// TIA Portal V17 export
// export: Created 2025-03-05T08:00:57.341892Z, ExportSetting WithDefaults, DisplayName Totally Integrated Automation Portal, DisplayVersion V17 Update 8, DisplayName TIA Portal Openness, DisplayVersion V17 Update 8, DisplayName TIA Portal Version Control Interface, DisplayVersion V17, DisplayName SINAMICS Startdrive Advanced, DisplayVersion V17 SP2, DisplayName SINAMICS Startdrive G110M, G120, G120C, G120D, G120P, G115D, DisplayVersion V17 SP2, DisplayName SINAMICS Startdrive G130, G150, S120, S150, SINAMICS MV, S210, DisplayVersion V17 SP2, DisplayName STEP 7 Professional, DisplayVersion V17 Update 8, DisplayName SINUMERIK ONE STEP 7 Toolbox, DisplayVersion V17 Update 12, DisplayName SINUMERIK 840D sl STEP 7 Toolbox, DisplayVersion V17 Update 12, DisplayName STEP 7 Safety, DisplayVersion V17 Update 6, DisplayName WinCC Advanced, DisplayVersion V17 Update 8
FUNCTION_BLOCK "FB1501_GENERAL_GAS_SYSTEM_VALVE"   // FB1501, LAD
{ S7_Optimized_Access := 'FALSE' }
AUTHOR : ETXETAR
VERSION : 1.0
// stored: AutoNumber false, IsIECCheckEnabled false, SetENOAutomatically false, UDAEnableTagReadback false
   VAR_INPUT
      PRESSURE : Bool;   // PRESSURE INPUT
      HMI_REQ_LINE : Bool;   // HMI REQUEST LINE
   END_VAR
   VAR_OUTPUT
      HMI_POWER_UP_COND_OFF : Bool;   // HMI POWER UP CONDITIONS OFF
      HMI_POWER_UP_COND_ON : Bool;   // HMI POWER UP CONDITIONS ON
      HMI_POWER_UP_EXECU_LEFT : Bool;   // HMI POWER UP EXECUTABLE LEFT
      HMI_POWER_UP_EXECU_RIGHT : Bool;   // HMI POWER UP EXECUTABLE RIGHT
      MAIN_VALVE : Bool;   // MAIN VALVE OUTPUT
   END_VAR
   VAR DB_SPECIFIC
      AIR_FLOW_VALUE : Real;   // AIR FLOW INPUT
      TEMPERATURE_VALUE : Real;   // TEMPERATURE INPUT VALUE
      PRESS_NOT_REACHED_ALARM : Bool;   // PRESSURE NOT REACHED ALARM
      PRESS_SWITCH_ALARM : Bool;   // PRESSURE SWITCH ALARM
      PRESS_MISSING_ALARM : Bool;   // PRESSURE MISSING ALARM
      CONNECTION_SENSOR_1_ALARM : Bool;   // CONNECTION SENSOR 1 ALARM
      CONNECTION_SENSOR_2_ALARM : Bool;   // CONNECTION SENSOR 2 ALARM
      UNBLOCK_DRIVE_PRESS_ALARM : Bool;   // UNBLOCK DRIVE PRESSURE ALARM
      UNBLOCK_DRIVE_PRESS_SWITCH_ALARM : Bool;   // UNBLOCK DRIVE PRESSURE SWITCH ALARM
      PRESSURIZATION_ALARM : Bool;   // PRESSURIZATION ALARM
      PRESSURIZATION_SWITCH_ALARM : Bool;   // PRESSURIZATION SWITCH ALARM
      PNEUMATIC_TEMPERATURE_INPUT_ALARM : Bool;   // PNEUMATIC INPUT TEMPERATURE ALARM
      PNEUMATIC_FLOW_INPUT_ALARM : Bool;   // PNEUMATIC INPUT FLOW ALARM
      U01_GRIPPER_PRESSURIZATION_ALARM : Bool;   // UNIT 01 GRIPPER PRESSURIZATION ALARM
      U01_GRIPPER_PRESSURIZATION_SWITCH_ALARM : Bool;   // UNIT 01 GRIPPER PRESSURIZATION SWITCH ALARM
      U01_LABERINT_PRESSURIZATION_ALARM : Bool;   // UNIT 01 LABERINT PRESSURIZATION ALARM
      U01_LABERINT_PRESSURIZATION_SWITCH_ALARM : Bool;   // UNIT 01 LABERINT PRESSURIZATION SWITCH ALARM
      U01_UPPER_TABLE_PRESSURIZATION_ALARM : Bool;   // UNIT 01 UPPER TABLE PRESSURIZATION ALARM
      U01_UPPER_TABLE_PRESSURIZATION_SWITCH_ALARM : Bool;   // UNIT 01 UPPER TABLE PRESSURIZATION SWITCH ALARM
      U01_LOWER_TABLE_PRESSURIZATION_ALARM : Bool;   // UNIT 01 LOWER TABLE PRESSURIZATION ALARM
      U01_LOWER_TABLE_PRESSURIZATION_SWITCH_ALARM : Bool;   // UNIT 01 LOWER TABLE PRESSURIZATION SWITCH ALARM
      U01_CART_AXIS_X_PRESSURIZATION_ALARM : Bool;   // UNIT 01 CART AXIS X PRESSURIZATION ALARM
      U01_CART_AXIS_X_PRESSURIZATION_SWITCH_ALARM : Bool;   // UNIT 01 CART AXIS X PRESSURIZATION SWITCH ALARM
      U01_STA_3_MEAS_PRESSURIZATION_ALARM : Bool;   // UNIT 01 STATION 3 MEASUREMENT UNIT PRESSURIZATION ALARM
      U01_STA_3_MEAS_PRESSURIZATION_SWITCH_ALARM : Bool;   // UNIT 01 STATION 3 MEASUREMENT UNIT PRESSURIZATION SWITCH ALARM
      U02_GRIPPER_PRESSURIZATION_ALARM : Bool;   // UNIT 02 GRIPPER PRESSURIZATION ALARM
      U02_GRIPPER_PRESSURIZATION_SWITCH_ALARM : Bool;   // UNIT 02 GRIPPER PRESSURIZATION SWITCH ALARM
      U02_LABERINT_PRESSURIZATION_ALARM : Bool;   // UNIT 02 LABERINT PRESSURIZATION ALARM
      U02_LABERINT_PRESSURIZATION_SWITCH_ALARM : Bool;   // UNIT 02 LABERINT PRESSURIZATION SWITCH ALARM
      U02_UPPER_TABLE_PRESSURIZATION_ALARM : Bool;   // UNIT 02 UPPER TABLE PRESSURIZATION ALARM
      U02_UPPER_TABLE_PRESSURIZATION_SWITCH_ALARM : Bool;   // UNIT 02 UPPER TABLE PRESSURIZATION SWITCH ALARM
      U02_LOWER_TABLE_PRESSURIZATION_ALARM : Bool;   // UNIT 02 LOWER TABLE PRESSURIZATION ALARM
      U02_LOWER_TABLE_PRESSURIZATION_SWITCH_ALARM : Bool;   // UNIT 02 LOWER TABLE PRESSURIZATION SWITCH ALARM
      U02_CART_AXIS_X_PRESSURIZATION_ALARM : Bool;   // UNIT 02 CART AXIS X PRESSURIZATION ALARM
      U02_CART_AXIS_X_PRESSURIZATION_SWITCH_ALARM : Bool;   // UNIT 02 CART AXIS X PRESSURIZATION SWITCH ALARM
      U02_STA_3_MEAS_PRESSURIZATION_ALARM : Bool;   // UNIT 02 STATION 3 MEASUREMENT UNIT PRESSURIZATION ALARM
      U02_STA_3_MEAS_PRESSURIZATION_SWITCH_ALARM : Bool;   // UNIT 02 STATION 3 MEASUREMENT UNIT PRESSURIZATION SWITCH ALARM
      SWITCH_ON_GENERAL_CONDITIONS : Bool;   // SWITCH ON GENERAL CONDITIONS
      SWITCH_ON_INITIAL_CONDITIONS : Bool;   // SWITCH ON INITIAL CONDITIONS
      SWITCH_ON_MANUAL_REQUEST : Bool;   // SWITCH ON MANUAL REQUEST
      SWITCH_ON_AUTO_REQUEST : Bool;   // SWITCH ON AUTO REQUEST
      SWITCH_ON_GLOBAL_REQUEST : Bool;   // SWITCH ON GLOBAL REQUEST
      SWITCH_ON_COMMAND : Bool;   // SWITCH ON COMMAND
      SWITCH_ON : Bool;   // SWITCH ON
      IN_SERVICE : Bool;   // IN SERVICE
      SWITCH_OFF_GENERAL_CONDITIONS : Bool;   // SWITCH OFF GENERAL CONDITIONS
      SWITCH_OFF_INITIAL_CONDITIONS : Bool;   // SWITCH OFF INITIAL CONDITIONS
      SWITCH_OFF_MANUAL_REQUEST : Bool;   // SWITCH OFF MANUAL REQUEST
      SWITCH_OFF_AUTO_REQUEST : Bool;   // SWITCH OFF AUTO REQUEST
      SWITCH_OFF_GLOBAL_REQUEST : Bool;   // SWITCH OFF GLOBAL REQUEST
      SWITCH_OFF_COMMAND : Bool;   // SWITCH OFF COMMAND
      SWITCH_OFF : Bool;   // SWITCH OFF
      OUT_OF_SERVICE : Bool;   // OUT OF SERVICE
      MANUAL_REQUEST_HELP : Bool;   // MANUAL REQUEST HELP
      SWITCH_ON_GENERAL_CONDITION_HELP : Bool;   // SWITCH ON GENERAL CONDITION HELP
      SWITCH_ON_INITIAL_CONDITION_HELP : Bool;   // SWITCH ON INITIAL CONDITION HELP
      SWITCH_OFF_GENERAL_CONDITION_HELP : Bool;   // SWITCH OFF GENERAL CONDITION HELP
      SWITCH_OFF_INITIAL_CONDITION_HELP : Bool;   // SWITCH OFF INITIAL CONDITION HELP
      ANY_ACTIVE_ALARM : Bool;   // ANY ACTIVE ALARM
      IS_ALARMS : Bool;   // IMMEDIATE STOP ALARMS
      SEOC_ALARMS : Bool;   // STOP END OF CYCLE ALARMS
      WARNINGS : Bool;   // WARNINGS
      WARNINGS_GONE : Bool;   // WARNINGS GONE
      TIMER_PRESSURE_ALARM : TON_TIME;   // PRESSURE TIMER
      TIMER_PRESSURE_SWITCH_ALARM : TON_TIME;   // PRESSURE SWITCH TIMER
      TIMER_PRESSURE_MISSING_ALARM : TON_TIME;   // PRESSURE MISSING TIMER
      TIMER_CONNECTION_SENSOR_1_ALARM : TON_TIME;   // CONNECTION SENSOR 1 TIMER
      TIMER_CONNECTION_SENSOR_1_SWITCH_ALARM : TON_TIME;   // CONNECTION SENSOR 1 SWITCH TIMER
      TIMER_CONNECTION_SENSOR_2_ALARM : TON_TIME;   // CONNECTION SENSOR 2 TIMER
      TIMER_CONNECTION_SENSOR_2_SWITCH_ALARM : TON_TIME;   // CONNECTION SENSOR 2 SWITCH TIMER
      TIMER_DRIVE_PRESSURE_UNBLOCK_ALARM : TON_TIME;   // DRIVE PRESSURE UNBLOCK TIMER
      TIMER_DRIVE_PRESSURE_UNBLOCK_SWITCH_ALARM : TON_TIME;   // DRIVE PRESSURE UNBLOCK SWITCH TIMER
      TIMER_PRESSURE_ON_DEVICES : TON_TIME;   // PRESSURE ON DEVICES TIMER
      TIMER_PRESSURE_OFF_DEVICES : TON_TIME;   // PRESSURE OFF DEVICES TIMER
      TIMER_PRESSURIZATION_OFF_DELAY { S7_SetPoint := 'True'} : TOF_TIME;
      PULSE { S7_SetPoint := 'True'} : Bool;
   END_VAR
   VAR_TEMP
      TEMPERATURE_TEMP : UInt;   // TEMPERATURE TEMPORAL
      PRESSURE_ON_DELAYED : Bool;   // PRESSURE ON DELAYED
      PRESSURE_OFF_DELAYED : Bool;   // PRESSURE OFF DELAYED
      DB_NUMBER : DInt;   // DB NUMBER FOR ALARM DECODING
   END_VAR
   // TIMER_PRESSURE_ALARM.PT := T#1M;
   // TIMER_PRESSURE_SWITCH_ALARM.PT := T#1M;
   // TIMER_PRESSURE_MISSING_ALARM.PT := T#1s;
   // TIMER_CONNECTION_SENSOR_1_ALARM.PT := T#1s;
   // TIMER_CONNECTION_SENSOR_1_SWITCH_ALARM.PT := T#1s;
   // TIMER_CONNECTION_SENSOR_2_ALARM.PT := T#1s;
   // TIMER_CONNECTION_SENSOR_2_SWITCH_ALARM.PT := T#1s;
   // TIMER_DRIVE_PRESSURE_UNBLOCK_ALARM.PT := T#3s;
   // TIMER_DRIVE_PRESSURE_UNBLOCK_SWITCH_ALARM.PT := T#3s;
   // TIMER_PRESSURE_ON_DEVICES.PT := T#5s;
   // TIMER_PRESSURE_OFF_DEVICES.PT := T#31M;
   // TIMER_PRESSURIZATION_OFF_DELAY.PT := T#30M;
   VAR_TEMP   // added for the SCL form of the ladder/FBD networks
      _w1 : Bool;
      _w2 : Bool;
   END_VAR
BEGIN

NETWORK
TITLE = READ INSTANCE DB
      L     DINO;
      +     10#800000;
      T     #DB_NUMBER;


REGION Network 2: SWITCH ON GENERAL CONDITIONS
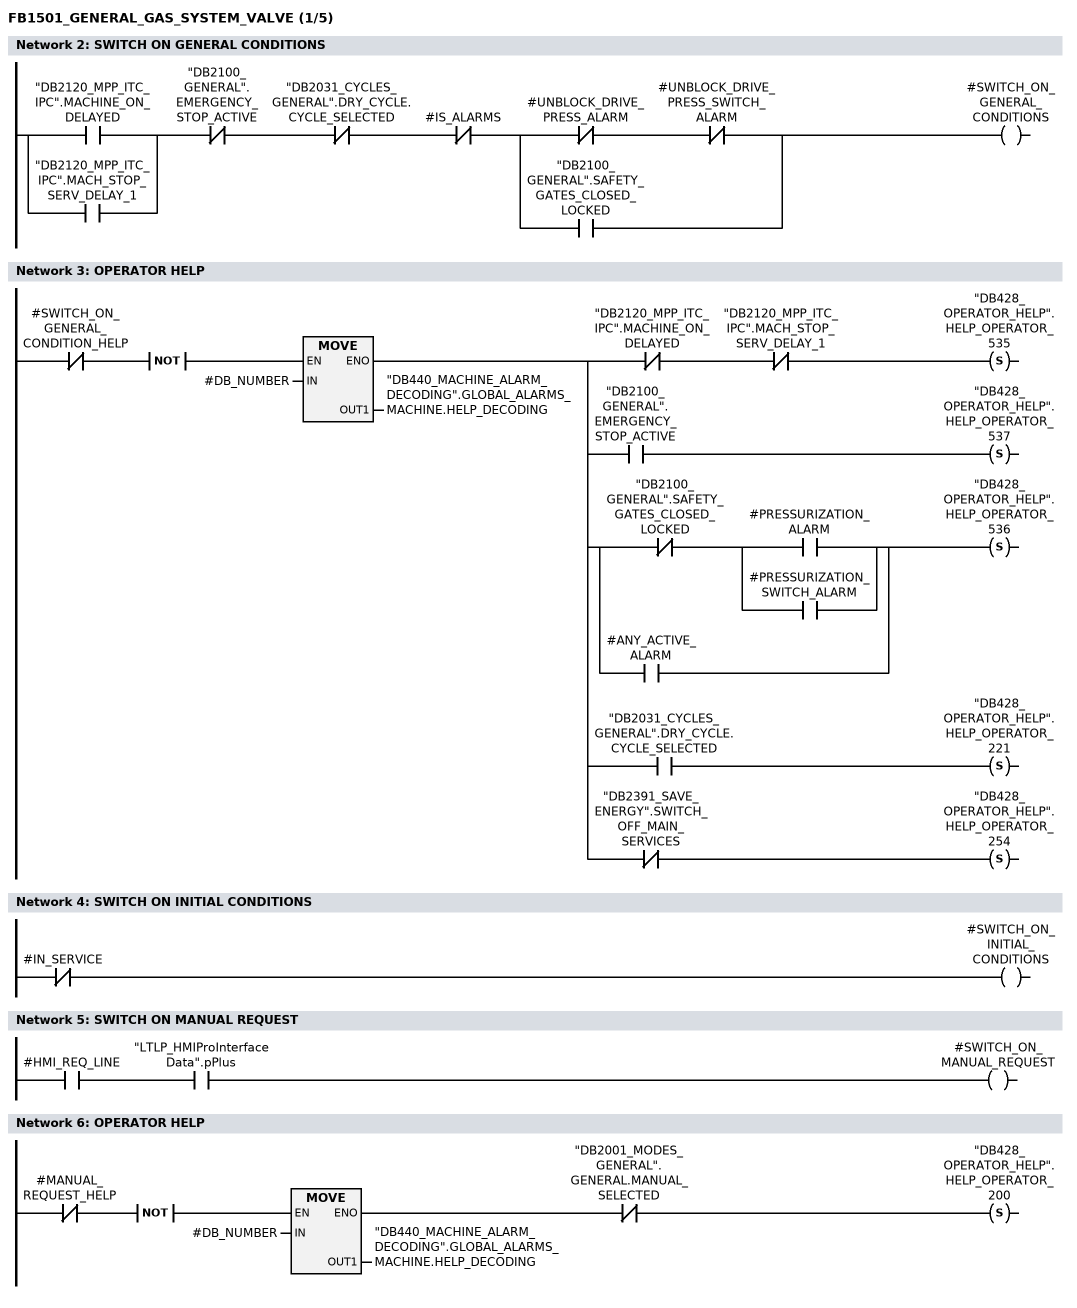
   RUNG wire#powerrail
      Contact( "DB2120_MPP_ITC_IPC".MACHINE_ON_DELAYED )
      wire#w1
      I_Contact( "DB2100_GENERAL".EMERGENCY_STOP_ACTIVE )
      I_Contact( "DB2031_CYCLES_GENERAL".DRY_CYCLE.CYCLE_SELECTED )
      I_Contact( #IS_ALARMS )
      wire#w2
      I_Contact( #UNBLOCK_DRIVE_PRESS_ALARM )
      I_Contact( #UNBLOCK_DRIVE_PRESS_SWITCH_ALARM )
      wire#w3
      Coil( #SWITCH_ON_GENERAL_CONDITIONS )
   END_RUNG
   RUNG wire#powerrail
      Contact( "DB2120_MPP_ITC_IPC".MACH_STOP_SERV_DELAY_1 )
   END_RUNG wire#w1
   RUNG wire#w2
      Contact( "DB2100_GENERAL".SAFETY_GATES_CLOSED_LOCKED )
   END_RUNG wire#w3
   // the same network as SCL:
   #SWITCH_ON_GENERAL_CONDITIONS := ("DB2120_MPP_ITC_IPC".MACHINE_ON_DELAYED OR "DB2120_MPP_ITC_IPC".MACH_STOP_SERV_DELAY_1) AND NOT "DB2100_GENERAL".EMERGENCY_STOP_ACTIVE AND NOT "DB2031_CYCLES_GENERAL".DRY_CYCLE.CYCLE_SELECTED AND NOT #IS_ALARMS AND ((NOT #UNBLOCK_DRIVE_PRESS_ALARM AND NOT #UNBLOCK_DRIVE_PRESS_SWITCH_ALARM) OR "DB2100_GENERAL".SAFETY_GATES_CLOSED_LOCKED);
END_REGION

REGION Network 3: OPERATOR HELP
   RUNG wire#powerrail
      I_Contact( #SWITCH_ON_GENERAL_CONDITION_HELP )
      Not()
      { S7_GenerateENO := "TRUE" } Move(in := #DB_NUMBER, out1 => "DB440_MACHINE_ALARM_DECODING".GLOBAL_ALARMS_MACHINE.HELP_DECODING)
      wire#w1
      I_Contact( "DB2120_MPP_ITC_IPC".MACHINE_ON_DELAYED )
      I_Contact( "DB2120_MPP_ITC_IPC".MACH_STOP_SERV_DELAY_1 )
      S_Coil( "DB428_OPERATOR_HELP".HELP_OPERATOR_535 )
   END_RUNG
   RUNG wire#w1
      Contact( "DB2100_GENERAL".EMERGENCY_STOP_ACTIVE )
      S_Coil( "DB428_OPERATOR_HELP".HELP_OPERATOR_537 )
   END_RUNG
   RUNG wire#w1
      I_Contact( "DB2100_GENERAL".SAFETY_GATES_CLOSED_LOCKED )
      wire#w2
      Contact( #PRESSURIZATION_ALARM )
      wire#w3
      S_Coil( "DB428_OPERATOR_HELP".HELP_OPERATOR_536 )
   END_RUNG
   RUNG wire#w2
      Contact( #PRESSURIZATION_SWITCH_ALARM )
   END_RUNG wire#w3
   RUNG wire#w1
      Contact( #ANY_ACTIVE_ALARM )
   END_RUNG wire#w3
   RUNG wire#w1
      Contact( "DB2031_CYCLES_GENERAL".DRY_CYCLE.CYCLE_SELECTED )
      S_Coil( "DB428_OPERATOR_HELP".HELP_OPERATOR_221 )
   END_RUNG
   RUNG wire#w1
      I_Contact( "DB2391_SAVE_ENERGY".SWITCH_OFF_MAIN_SERVICES )
      S_Coil( "DB428_OPERATOR_HELP".HELP_OPERATOR_254 )
   END_RUNG
   // the same network as SCL:
   // ENO of a box is taken as its EN; it also drops when the box reports an error
   #_w1 := NOT (NOT #SWITCH_ON_GENERAL_CONDITION_HELP);
   IF #_w1 THEN "DB440_MACHINE_ALARM_DECODING".GLOBAL_ALARMS_MACHINE.HELP_DECODING := #DB_NUMBER; END_IF;
   IF #_w1 AND NOT "DB2120_MPP_ITC_IPC".MACHINE_ON_DELAYED AND NOT "DB2120_MPP_ITC_IPC".MACH_STOP_SERV_DELAY_1 THEN
       "DB428_OPERATOR_HELP".HELP_OPERATOR_535 := TRUE;
   END_IF;
   IF #_w1 AND "DB2100_GENERAL".EMERGENCY_STOP_ACTIVE THEN
       "DB428_OPERATOR_HELP".HELP_OPERATOR_537 := TRUE;
   END_IF;
   IF #_w1 AND ((NOT "DB2100_GENERAL".SAFETY_GATES_CLOSED_LOCKED AND (#PRESSURIZATION_ALARM OR #PRESSURIZATION_SWITCH_ALARM)) OR #ANY_ACTIVE_ALARM) THEN
       "DB428_OPERATOR_HELP".HELP_OPERATOR_536 := TRUE;
   END_IF;
   IF #_w1 AND "DB2031_CYCLES_GENERAL".DRY_CYCLE.CYCLE_SELECTED THEN
       "DB428_OPERATOR_HELP".HELP_OPERATOR_221 := TRUE;
   END_IF;
   IF #_w1 AND NOT "DB2391_SAVE_ENERGY".SWITCH_OFF_MAIN_SERVICES THEN
       "DB428_OPERATOR_HELP".HELP_OPERATOR_254 := TRUE;
   END_IF;
END_REGION

REGION Network 4: SWITCH ON INITIAL CONDITIONS
   RUNG wire#powerrail
      I_Contact( #IN_SERVICE )
      Coil( #SWITCH_ON_INITIAL_CONDITIONS )
   END_RUNG
   // the same network as SCL:
   #SWITCH_ON_INITIAL_CONDITIONS := NOT #IN_SERVICE;
END_REGION

REGION Network 5: SWITCH ON MANUAL REQUEST
   RUNG wire#powerrail
      Contact( #HMI_REQ_LINE )
      Contact( "LTLP_HMIProInterfaceData".pPlus )
      Coil( #SWITCH_ON_MANUAL_REQUEST )
   END_RUNG
   // the same network as SCL:
   #SWITCH_ON_MANUAL_REQUEST := #HMI_REQ_LINE AND "LTLP_HMIProInterfaceData".pPlus;
END_REGION

REGION Network 6: OPERATOR HELP
   RUNG wire#powerrail
      I_Contact( #MANUAL_REQUEST_HELP )
      Not()
      { S7_GenerateENO := "TRUE" } Move(in := #DB_NUMBER, out1 => "DB440_MACHINE_ALARM_DECODING".GLOBAL_ALARMS_MACHINE.HELP_DECODING)
      I_Contact( "DB2001_MODES_GENERAL".GENERAL.MANUAL_SELECTED )
      S_Coil( "DB428_OPERATOR_HELP".HELP_OPERATOR_200 )
   END_RUNG
   // the same network as SCL:
   // ENO of a box is taken as its EN; it also drops when the box reports an error
   #_w1 := NOT (NOT #MANUAL_REQUEST_HELP);
   IF #_w1 THEN "DB440_MACHINE_ALARM_DECODING".GLOBAL_ALARMS_MACHINE.HELP_DECODING := #DB_NUMBER; END_IF;
   IF #_w1 AND NOT "DB2001_MODES_GENERAL".GENERAL.MANUAL_SELECTED THEN
       "DB428_OPERATOR_HELP".HELP_OPERATOR_200 := TRUE;
   END_IF;
END_REGION

REGION Network 7: SWITCH ON AUTO REQUEST
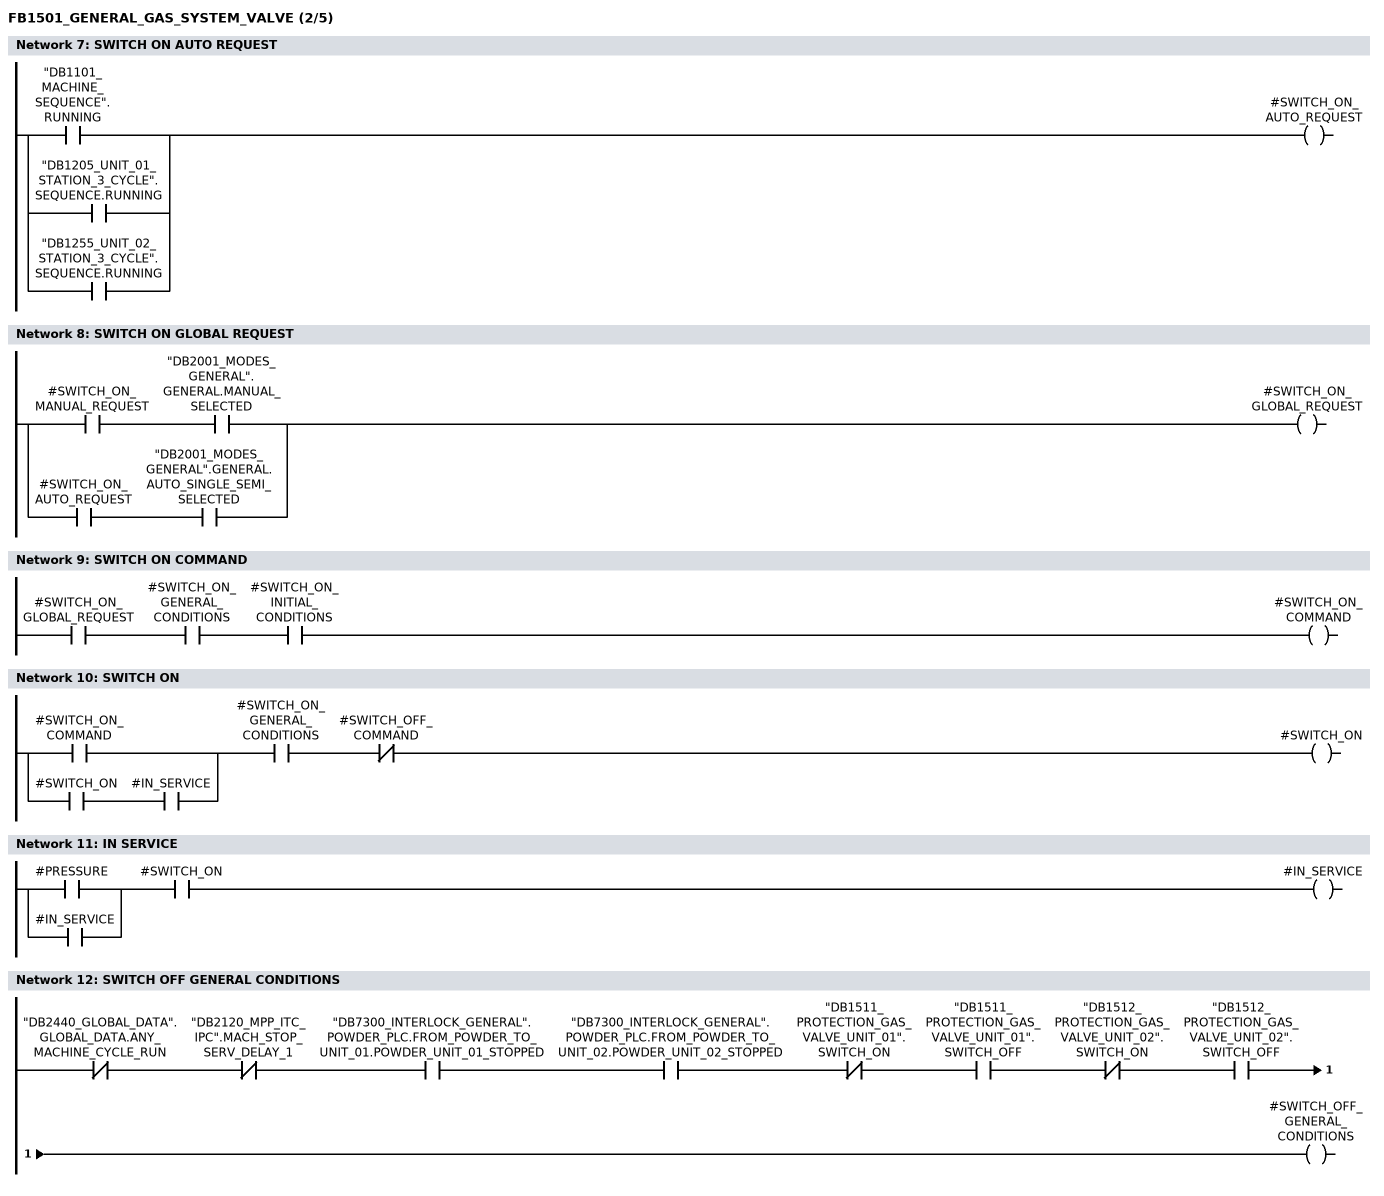
   RUNG wire#powerrail
      Contact( "DB1101_MACHINE_SEQUENCE".RUNNING )
      wire#w1
      Coil( #SWITCH_ON_AUTO_REQUEST )
   END_RUNG
   RUNG wire#powerrail
      Contact( "DB1205_UNIT_01_STATION_3_CYCLE".SEQUENCE.RUNNING )
   END_RUNG wire#w1
   RUNG wire#powerrail
      Contact( "DB1255_UNIT_02_STATION_3_CYCLE".SEQUENCE.RUNNING )
   END_RUNG wire#w1
   // the same network as SCL:
   #SWITCH_ON_AUTO_REQUEST := "DB1101_MACHINE_SEQUENCE".RUNNING OR "DB1205_UNIT_01_STATION_3_CYCLE".SEQUENCE.RUNNING OR "DB1255_UNIT_02_STATION_3_CYCLE".SEQUENCE.RUNNING;
END_REGION

REGION Network 8: SWITCH ON GLOBAL REQUEST
   RUNG wire#powerrail
      Contact( #SWITCH_ON_MANUAL_REQUEST )
      Contact( "DB2001_MODES_GENERAL".GENERAL.MANUAL_SELECTED )
      wire#w1
      Coil( #SWITCH_ON_GLOBAL_REQUEST )
   END_RUNG
   RUNG wire#powerrail
      Contact( #SWITCH_ON_AUTO_REQUEST )
      Contact( "DB2001_MODES_GENERAL".GENERAL.AUTO_SINGLE_SEMI_SELECTED )
   END_RUNG wire#w1
   // the same network as SCL:
   #SWITCH_ON_GLOBAL_REQUEST := (#SWITCH_ON_MANUAL_REQUEST AND "DB2001_MODES_GENERAL".GENERAL.MANUAL_SELECTED) OR (#SWITCH_ON_AUTO_REQUEST AND "DB2001_MODES_GENERAL".GENERAL.AUTO_SINGLE_SEMI_SELECTED);
END_REGION

REGION Network 9: SWITCH ON COMMAND
   RUNG wire#powerrail
      Contact( #SWITCH_ON_GLOBAL_REQUEST )
      Contact( #SWITCH_ON_GENERAL_CONDITIONS )
      Contact( #SWITCH_ON_INITIAL_CONDITIONS )
      Coil( #SWITCH_ON_COMMAND )
   END_RUNG
   // the same network as SCL:
   #SWITCH_ON_COMMAND := #SWITCH_ON_GLOBAL_REQUEST AND #SWITCH_ON_GENERAL_CONDITIONS AND #SWITCH_ON_INITIAL_CONDITIONS;
END_REGION

REGION Network 10: SWITCH ON
   RUNG wire#powerrail
      Contact( #SWITCH_ON_COMMAND )
      wire#w1
      Contact( #SWITCH_ON_GENERAL_CONDITIONS )
      I_Contact( #SWITCH_OFF_COMMAND )
      Coil( #SWITCH_ON )
   END_RUNG
   RUNG wire#powerrail
      Contact( #SWITCH_ON )
      Contact( #IN_SERVICE )
   END_RUNG wire#w1
   // the same network as SCL:
   #SWITCH_ON := (#SWITCH_ON_COMMAND OR (#SWITCH_ON AND #IN_SERVICE)) AND #SWITCH_ON_GENERAL_CONDITIONS AND NOT #SWITCH_OFF_COMMAND;
END_REGION

REGION Network 11: IN SERVICE
   RUNG wire#powerrail
      Contact( #PRESSURE )
      wire#w1
      Contact( #SWITCH_ON )
      Coil( #IN_SERVICE )
   END_RUNG
   RUNG wire#powerrail
      Contact( #IN_SERVICE )
   END_RUNG wire#w1
   // the same network as SCL:
   #IN_SERVICE := (#PRESSURE OR #IN_SERVICE) AND #SWITCH_ON;
END_REGION

REGION Network 12: SWITCH OFF GENERAL CONDITIONS
   RUNG wire#powerrail
      I_Contact( "DB2440_GLOBAL_DATA".GLOBAL_DATA.ANY_MACHINE_CYCLE_RUN )
      I_Contact( "DB2120_MPP_ITC_IPC".MACH_STOP_SERV_DELAY_1 )
      Contact( "DB7300_INTERLOCK_GENERAL".POWDER_PLC.FROM_POWDER_TO_UNIT_01.POWDER_UNIT_01_STOPPED )
      Contact( "DB7300_INTERLOCK_GENERAL".POWDER_PLC.FROM_POWDER_TO_UNIT_02.POWDER_UNIT_02_STOPPED )
      I_Contact( "DB1511_PROTECTION_GAS_VALVE_UNIT_01".SWITCH_ON )
      Contact( "DB1511_PROTECTION_GAS_VALVE_UNIT_01".SWITCH_OFF )
      I_Contact( "DB1512_PROTECTION_GAS_VALVE_UNIT_02".SWITCH_ON )
      Contact( "DB1512_PROTECTION_GAS_VALVE_UNIT_02".SWITCH_OFF )
      Coil( #SWITCH_OFF_GENERAL_CONDITIONS )
   END_RUNG
   // the same network as SCL:
   #SWITCH_OFF_GENERAL_CONDITIONS := NOT "DB2440_GLOBAL_DATA".GLOBAL_DATA.ANY_MACHINE_CYCLE_RUN AND NOT "DB2120_MPP_ITC_IPC".MACH_STOP_SERV_DELAY_1 AND "DB7300_INTERLOCK_GENERAL".POWDER_PLC.FROM_POWDER_TO_UNIT_01.POWDER_UNIT_01_STOPPED AND "DB7300_INTERLOCK_GENERAL".POWDER_PLC.FROM_POWDER_TO_UNIT_02.POWDER_UNIT_02_STOPPED AND NOT "DB1511_PROTECTION_GAS_VALVE_UNIT_01".SWITCH_ON AND "DB1511_PROTECTION_GAS_VALVE_UNIT_01".SWITCH_OFF AND NOT "DB1512_PROTECTION_GAS_VALVE_UNIT_02".SWITCH_ON AND "DB1512_PROTECTION_GAS_VALVE_UNIT_02".SWITCH_OFF;
END_REGION

REGION Network 13: OPERATOR HELP
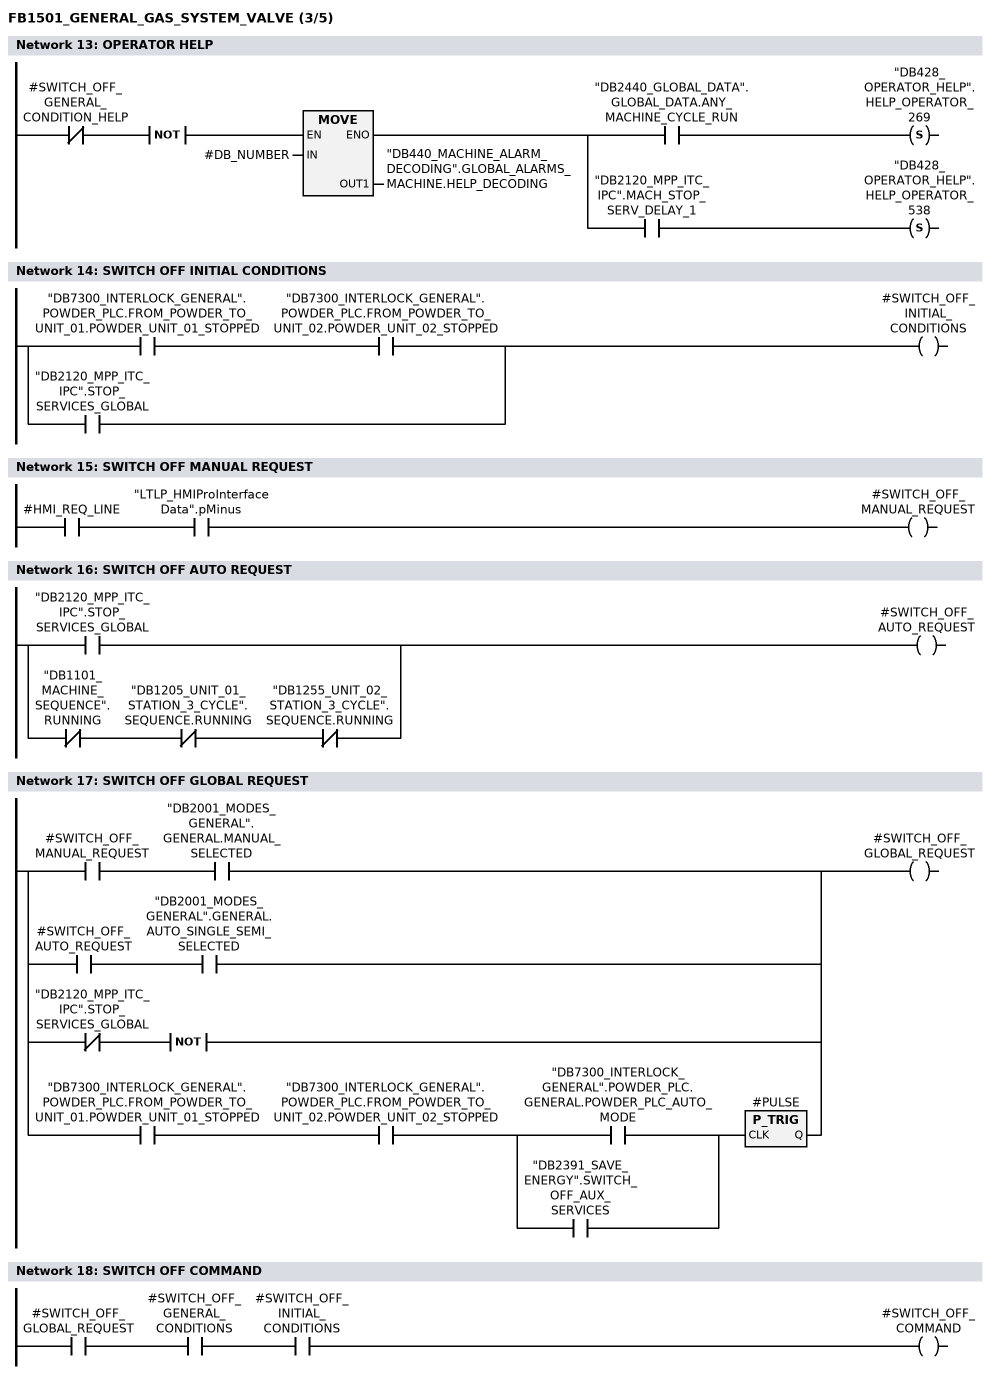
   RUNG wire#powerrail
      I_Contact( #SWITCH_OFF_GENERAL_CONDITION_HELP )
      Not()
      { S7_GenerateENO := "TRUE" } Move(in := #DB_NUMBER, out1 => "DB440_MACHINE_ALARM_DECODING".GLOBAL_ALARMS_MACHINE.HELP_DECODING)
      wire#w1
      Contact( "DB2440_GLOBAL_DATA".GLOBAL_DATA.ANY_MACHINE_CYCLE_RUN )
      S_Coil( "DB428_OPERATOR_HELP".HELP_OPERATOR_269 )
   END_RUNG
   RUNG wire#w1
      Contact( "DB2120_MPP_ITC_IPC".MACH_STOP_SERV_DELAY_1 )
      S_Coil( "DB428_OPERATOR_HELP".HELP_OPERATOR_538 )
   END_RUNG
   // the same network as SCL:
   // ENO of a box is taken as its EN; it also drops when the box reports an error
   #_w1 := NOT (NOT #SWITCH_OFF_GENERAL_CONDITION_HELP);
   IF #_w1 THEN "DB440_MACHINE_ALARM_DECODING".GLOBAL_ALARMS_MACHINE.HELP_DECODING := #DB_NUMBER; END_IF;
   IF #_w1 AND "DB2440_GLOBAL_DATA".GLOBAL_DATA.ANY_MACHINE_CYCLE_RUN THEN
       "DB428_OPERATOR_HELP".HELP_OPERATOR_269 := TRUE;
   END_IF;
   IF #_w1 AND "DB2120_MPP_ITC_IPC".MACH_STOP_SERV_DELAY_1 THEN
       "DB428_OPERATOR_HELP".HELP_OPERATOR_538 := TRUE;
   END_IF;
END_REGION

REGION Network 14: SWITCH OFF INITIAL CONDITIONS
   RUNG wire#powerrail
      Contact( "DB7300_INTERLOCK_GENERAL".POWDER_PLC.FROM_POWDER_TO_UNIT_01.POWDER_UNIT_01_STOPPED )
      Contact( "DB7300_INTERLOCK_GENERAL".POWDER_PLC.FROM_POWDER_TO_UNIT_02.POWDER_UNIT_02_STOPPED )
      wire#w1
      Coil( #SWITCH_OFF_INITIAL_CONDITIONS )
   END_RUNG
   RUNG wire#powerrail
      Contact( "DB2120_MPP_ITC_IPC".STOP_SERVICES_GLOBAL )
   END_RUNG wire#w1
   // the same network as SCL:
   #SWITCH_OFF_INITIAL_CONDITIONS := ("DB7300_INTERLOCK_GENERAL".POWDER_PLC.FROM_POWDER_TO_UNIT_01.POWDER_UNIT_01_STOPPED AND "DB7300_INTERLOCK_GENERAL".POWDER_PLC.FROM_POWDER_TO_UNIT_02.POWDER_UNIT_02_STOPPED) OR "DB2120_MPP_ITC_IPC".STOP_SERVICES_GLOBAL;
END_REGION

REGION Network 15: SWITCH OFF MANUAL REQUEST
   RUNG wire#powerrail
      Contact( #HMI_REQ_LINE )
      Contact( "LTLP_HMIProInterfaceData".pMinus )
      Coil( #SWITCH_OFF_MANUAL_REQUEST )
   END_RUNG
   // the same network as SCL:
   #SWITCH_OFF_MANUAL_REQUEST := #HMI_REQ_LINE AND "LTLP_HMIProInterfaceData".pMinus;
END_REGION

REGION Network 16: SWITCH OFF AUTO REQUEST
   RUNG wire#powerrail
      Contact( "DB2120_MPP_ITC_IPC".STOP_SERVICES_GLOBAL )
      wire#w1
      Coil( #SWITCH_OFF_AUTO_REQUEST )
   END_RUNG
   RUNG wire#powerrail
      I_Contact( "DB1101_MACHINE_SEQUENCE".RUNNING )
      I_Contact( "DB1205_UNIT_01_STATION_3_CYCLE".SEQUENCE.RUNNING )
      I_Contact( "DB1255_UNIT_02_STATION_3_CYCLE".SEQUENCE.RUNNING )
   END_RUNG wire#w1
   // the same network as SCL:
   #SWITCH_OFF_AUTO_REQUEST := "DB2120_MPP_ITC_IPC".STOP_SERVICES_GLOBAL OR (NOT "DB1101_MACHINE_SEQUENCE".RUNNING AND NOT "DB1205_UNIT_01_STATION_3_CYCLE".SEQUENCE.RUNNING AND NOT "DB1255_UNIT_02_STATION_3_CYCLE".SEQUENCE.RUNNING);
END_REGION

REGION Network 17: SWITCH OFF GLOBAL REQUEST
   RUNG wire#powerrail
      Contact( #SWITCH_OFF_MANUAL_REQUEST )
      Contact( "DB2001_MODES_GENERAL".GENERAL.MANUAL_SELECTED )
      wire#w1
      Coil( #SWITCH_OFF_GLOBAL_REQUEST )
   END_RUNG
   RUNG wire#powerrail
      Contact( #SWITCH_OFF_AUTO_REQUEST )
      Contact( "DB2001_MODES_GENERAL".GENERAL.AUTO_SINGLE_SEMI_SELECTED )
   END_RUNG wire#w1
   RUNG wire#powerrail
      I_Contact( "DB2120_MPP_ITC_IPC".STOP_SERVICES_GLOBAL )
      Not()
   END_RUNG wire#w1
   RUNG wire#powerrail
      Contact( "DB7300_INTERLOCK_GENERAL".POWDER_PLC.FROM_POWDER_TO_UNIT_01.POWDER_UNIT_01_STOPPED )
      Contact( "DB7300_INTERLOCK_GENERAL".POWDER_PLC.FROM_POWDER_TO_UNIT_02.POWDER_UNIT_02_STOPPED )
      wire#w2
      Contact( "DB7300_INTERLOCK_GENERAL".POWDER_PLC.GENERAL.POWDER_PLC_AUTO_MODE )
      wire#w3
      P_Trig( #PULSE )
   END_RUNG wire#w1
   RUNG wire#w2
      Contact( "DB2391_SAVE_ENERGY".SWITCH_OFF_AUX_SERVICES )
   END_RUNG wire#w3
   // the same network as SCL:
   #_w1 := "DB7300_INTERLOCK_GENERAL".POWDER_PLC.FROM_POWDER_TO_UNIT_01.POWDER_UNIT_01_STOPPED AND "DB7300_INTERLOCK_GENERAL".POWDER_PLC.FROM_POWDER_TO_UNIT_02.POWDER_UNIT_02_STOPPED AND ("DB7300_INTERLOCK_GENERAL".POWDER_PLC.GENERAL.POWDER_PLC_AUTO_MODE OR "DB2391_SAVE_ENERGY".SWITCH_OFF_AUX_SERVICES);
   #_w2 := #_w1 AND NOT #PULSE;   // rising edge
   #PULSE := #_w1;
   #SWITCH_OFF_GLOBAL_REQUEST := (#SWITCH_OFF_MANUAL_REQUEST AND "DB2001_MODES_GENERAL".GENERAL.MANUAL_SELECTED) OR (#SWITCH_OFF_AUTO_REQUEST AND "DB2001_MODES_GENERAL".GENERAL.AUTO_SINGLE_SEMI_SELECTED) OR NOT (NOT "DB2120_MPP_ITC_IPC".STOP_SERVICES_GLOBAL) OR #_w2;
END_REGION

REGION Network 18: SWITCH OFF COMMAND
   RUNG wire#powerrail
      Contact( #SWITCH_OFF_GLOBAL_REQUEST )
      Contact( #SWITCH_OFF_GENERAL_CONDITIONS )
      Contact( #SWITCH_OFF_INITIAL_CONDITIONS )
      Coil( #SWITCH_OFF_COMMAND )
   END_RUNG
   // the same network as SCL:
   #SWITCH_OFF_COMMAND := #SWITCH_OFF_GLOBAL_REQUEST AND #SWITCH_OFF_GENERAL_CONDITIONS AND #SWITCH_OFF_INITIAL_CONDITIONS;
END_REGION

REGION Network 19: OUT OF SERVICE
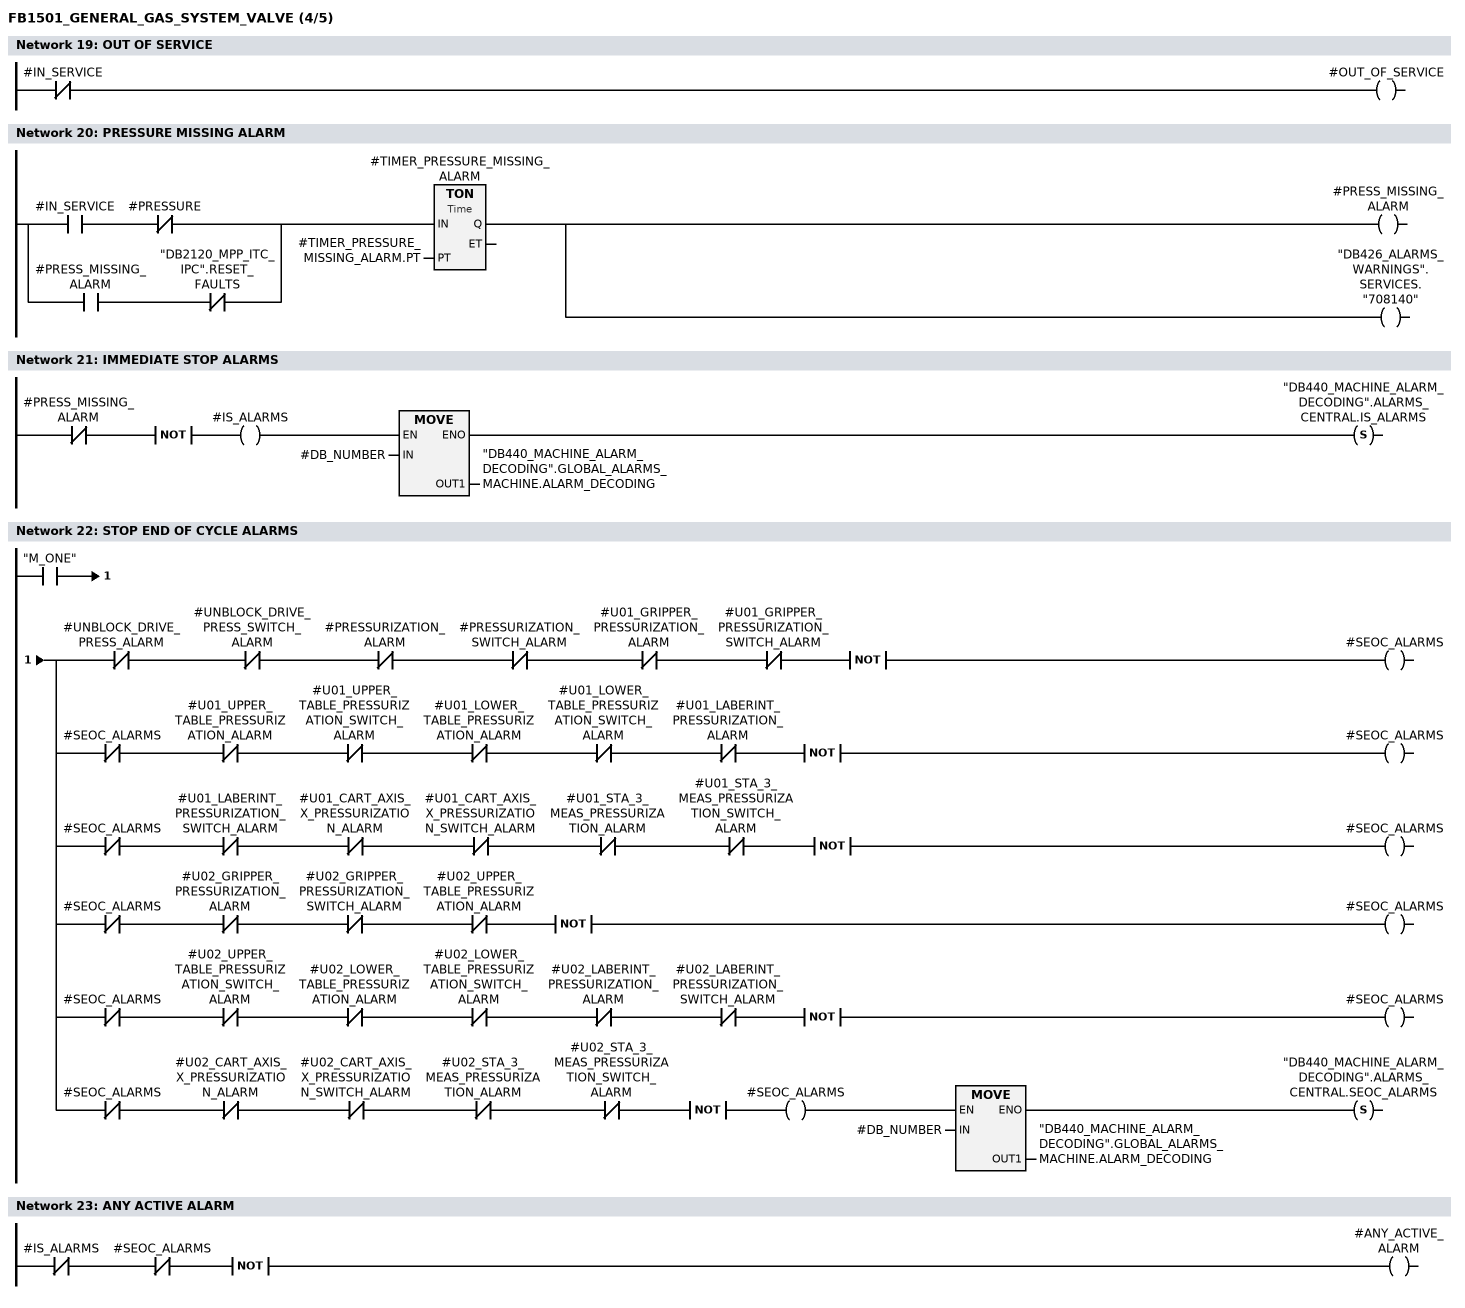
   RUNG wire#powerrail
      I_Contact( #IN_SERVICE )
      Coil( #OUT_OF_SERVICE )
   END_RUNG
   // the same network as SCL:
   #OUT_OF_SERVICE := NOT #IN_SERVICE;
END_REGION

REGION Network 20: PRESSURE MISSING ALARM
   RUNG wire#powerrail
      Contact( #IN_SERVICE )
      I_Contact( #PRESSURE )
      wire#w1
      { S7_Templates := "time_type := Time" } #TIMER_PRESSURE_MISSING_ALARM.TON(pt := #TIMER_PRESSURE_MISSING_ALARM.PT, et =>)
      wire#w2
      Coil( #PRESS_MISSING_ALARM )
   END_RUNG
   RUNG wire#powerrail
      Contact( #PRESS_MISSING_ALARM )
      I_Contact( "DB2120_MPP_ITC_IPC".RESET_FAULTS )
   END_RUNG wire#w1
   RUNG wire#w2
      Coil( "DB426_ALARMS_WARNINGS".SERVICES."708140" )
   END_RUNG
   // the same network as SCL:
   #TIMER_PRESSURE_MISSING_ALARM(IN := (#IN_SERVICE AND NOT #PRESSURE) OR (#PRESS_MISSING_ALARM AND NOT "DB2120_MPP_ITC_IPC".RESET_FAULTS),   // TON
                           PT := #TIMER_PRESSURE_MISSING_ALARM.PT);
   #PRESS_MISSING_ALARM := #TIMER_PRESSURE_MISSING_ALARM.Q;
   "DB426_ALARMS_WARNINGS".SERVICES."708140" := #TIMER_PRESSURE_MISSING_ALARM.Q;
END_REGION

REGION Network 21: IMMEDIATE STOP ALARMS
   RUNG wire#powerrail
      I_Contact( #PRESS_MISSING_ALARM )
      Not()
      Coil( #IS_ALARMS )
      Move(in := #DB_NUMBER, out1 => "DB440_MACHINE_ALARM_DECODING".GLOBAL_ALARMS_MACHINE.ALARM_DECODING)
      S_Coil( "DB440_MACHINE_ALARM_DECODING".ALARMS_CENTRAL.IS_ALARMS )
   END_RUNG
   // the same network as SCL:
   #IS_ALARMS := NOT (NOT #PRESS_MISSING_ALARM);
   IF NOT (NOT #PRESS_MISSING_ALARM) THEN
       "DB440_MACHINE_ALARM_DECODING".GLOBAL_ALARMS_MACHINE.ALARM_DECODING := #DB_NUMBER;
       "DB440_MACHINE_ALARM_DECODING".ALARMS_CENTRAL.IS_ALARMS := TRUE;
   END_IF;
END_REGION

REGION Network 22: STOP END OF CYCLE ALARMS
   RUNG wire#powerrail
      Contact( "M_ONE" )
      wire#w1
      I_Contact( #UNBLOCK_DRIVE_PRESS_ALARM )
      I_Contact( #UNBLOCK_DRIVE_PRESS_SWITCH_ALARM )
      I_Contact( #PRESSURIZATION_ALARM )
      I_Contact( #PRESSURIZATION_SWITCH_ALARM )
      I_Contact( #U01_GRIPPER_PRESSURIZATION_ALARM )
      I_Contact( #U01_GRIPPER_PRESSURIZATION_SWITCH_ALARM )
      Not()
      Coil( #SEOC_ALARMS )
   END_RUNG
   RUNG wire#w1
      I_Contact( #SEOC_ALARMS )
      I_Contact( #U01_UPPER_TABLE_PRESSURIZATION_ALARM )
      I_Contact( #U01_UPPER_TABLE_PRESSURIZATION_SWITCH_ALARM )
      I_Contact( #U01_LOWER_TABLE_PRESSURIZATION_ALARM )
      I_Contact( #U01_LOWER_TABLE_PRESSURIZATION_SWITCH_ALARM )
      I_Contact( #U01_LABERINT_PRESSURIZATION_ALARM )
      Not()
      Coil( #SEOC_ALARMS )
   END_RUNG
   RUNG wire#w1
      I_Contact( #SEOC_ALARMS )
      I_Contact( #U01_LABERINT_PRESSURIZATION_SWITCH_ALARM )
      I_Contact( #U01_CART_AXIS_X_PRESSURIZATION_ALARM )
      I_Contact( #U01_CART_AXIS_X_PRESSURIZATION_SWITCH_ALARM )
      I_Contact( #U01_STA_3_MEAS_PRESSURIZATION_ALARM )
      I_Contact( #U01_STA_3_MEAS_PRESSURIZATION_SWITCH_ALARM )
      Not()
      Coil( #SEOC_ALARMS )
   END_RUNG
   RUNG wire#w1
      I_Contact( #SEOC_ALARMS )
      I_Contact( #U02_GRIPPER_PRESSURIZATION_ALARM )
      I_Contact( #U02_GRIPPER_PRESSURIZATION_SWITCH_ALARM )
      I_Contact( #U02_UPPER_TABLE_PRESSURIZATION_ALARM )
      Not()
      Coil( #SEOC_ALARMS )
   END_RUNG
   RUNG wire#w1
      I_Contact( #SEOC_ALARMS )
      I_Contact( #U02_UPPER_TABLE_PRESSURIZATION_SWITCH_ALARM )
      I_Contact( #U02_LOWER_TABLE_PRESSURIZATION_ALARM )
      I_Contact( #U02_LOWER_TABLE_PRESSURIZATION_SWITCH_ALARM )
      I_Contact( #U02_LABERINT_PRESSURIZATION_ALARM )
      I_Contact( #U02_LABERINT_PRESSURIZATION_SWITCH_ALARM )
      Not()
      Coil( #SEOC_ALARMS )
   END_RUNG
   RUNG wire#w1
      I_Contact( #SEOC_ALARMS )
      I_Contact( #U02_CART_AXIS_X_PRESSURIZATION_ALARM )
      I_Contact( #U02_CART_AXIS_X_PRESSURIZATION_SWITCH_ALARM )
      I_Contact( #U02_STA_3_MEAS_PRESSURIZATION_ALARM )
      I_Contact( #U02_STA_3_MEAS_PRESSURIZATION_SWITCH_ALARM )
      Not()
      Coil( #SEOC_ALARMS )
      Move(in := #DB_NUMBER, out1 => "DB440_MACHINE_ALARM_DECODING".GLOBAL_ALARMS_MACHINE.ALARM_DECODING)
      S_Coil( "DB440_MACHINE_ALARM_DECODING".ALARMS_CENTRAL.SEOC_ALARMS )
   END_RUNG
   // the same network as SCL:
   #SEOC_ALARMS := NOT ("M_ONE" AND NOT #UNBLOCK_DRIVE_PRESS_ALARM AND NOT #UNBLOCK_DRIVE_PRESS_SWITCH_ALARM AND NOT #PRESSURIZATION_ALARM AND NOT #PRESSURIZATION_SWITCH_ALARM AND NOT #U01_GRIPPER_PRESSURIZATION_ALARM AND NOT #U01_GRIPPER_PRESSURIZATION_SWITCH_ALARM);
   #SEOC_ALARMS := NOT ("M_ONE" AND NOT #SEOC_ALARMS AND NOT #U01_UPPER_TABLE_PRESSURIZATION_ALARM AND NOT #U01_UPPER_TABLE_PRESSURIZATION_SWITCH_ALARM AND NOT #U01_LOWER_TABLE_PRESSURIZATION_ALARM AND NOT #U01_LOWER_TABLE_PRESSURIZATION_SWITCH_ALARM AND NOT #U01_LABERINT_PRESSURIZATION_ALARM);
   #SEOC_ALARMS := NOT ("M_ONE" AND NOT #SEOC_ALARMS AND NOT #U01_LABERINT_PRESSURIZATION_SWITCH_ALARM AND NOT #U01_CART_AXIS_X_PRESSURIZATION_ALARM AND NOT #U01_CART_AXIS_X_PRESSURIZATION_SWITCH_ALARM AND NOT #U01_STA_3_MEAS_PRESSURIZATION_ALARM AND NOT #U01_STA_3_MEAS_PRESSURIZATION_SWITCH_ALARM);
   #SEOC_ALARMS := NOT ("M_ONE" AND NOT #SEOC_ALARMS AND NOT #U02_GRIPPER_PRESSURIZATION_ALARM AND NOT #U02_GRIPPER_PRESSURIZATION_SWITCH_ALARM AND NOT #U02_UPPER_TABLE_PRESSURIZATION_ALARM);
   #SEOC_ALARMS := NOT ("M_ONE" AND NOT #SEOC_ALARMS AND NOT #U02_UPPER_TABLE_PRESSURIZATION_SWITCH_ALARM AND NOT #U02_LOWER_TABLE_PRESSURIZATION_ALARM AND NOT #U02_LOWER_TABLE_PRESSURIZATION_SWITCH_ALARM AND NOT #U02_LABERINT_PRESSURIZATION_ALARM AND NOT #U02_LABERINT_PRESSURIZATION_SWITCH_ALARM);
   #SEOC_ALARMS := NOT ("M_ONE" AND NOT #SEOC_ALARMS AND NOT #U02_CART_AXIS_X_PRESSURIZATION_ALARM AND NOT #U02_CART_AXIS_X_PRESSURIZATION_SWITCH_ALARM AND NOT #U02_STA_3_MEAS_PRESSURIZATION_ALARM AND NOT #U02_STA_3_MEAS_PRESSURIZATION_SWITCH_ALARM);
   IF #SEOC_ALARMS THEN
       "DB440_MACHINE_ALARM_DECODING".GLOBAL_ALARMS_MACHINE.ALARM_DECODING := #DB_NUMBER;
       "DB440_MACHINE_ALARM_DECODING".ALARMS_CENTRAL.SEOC_ALARMS := TRUE;
   END_IF;
END_REGION

REGION Network 23: ANY ACTIVE ALARM
   RUNG wire#powerrail
      I_Contact( #IS_ALARMS )
      I_Contact( #SEOC_ALARMS )
      Not()
      Coil( #ANY_ACTIVE_ALARM )
   END_RUNG
   // the same network as SCL:
   #ANY_ACTIVE_ALARM := NOT (NOT #IS_ALARMS AND NOT #SEOC_ALARMS);
END_REGION

REGION Network 24: MANUAL REQUEST HELP
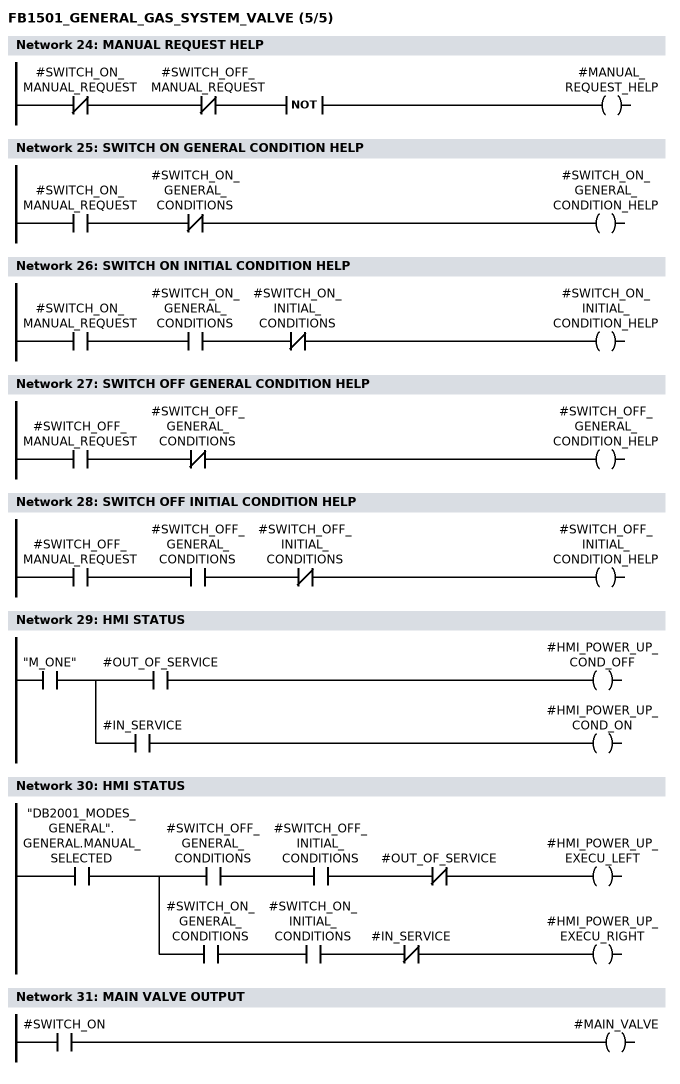
   RUNG wire#powerrail
      I_Contact( #SWITCH_ON_MANUAL_REQUEST )
      I_Contact( #SWITCH_OFF_MANUAL_REQUEST )
      Not()
      Coil( #MANUAL_REQUEST_HELP )
   END_RUNG
   // the same network as SCL:
   #MANUAL_REQUEST_HELP := NOT (NOT #SWITCH_ON_MANUAL_REQUEST AND NOT #SWITCH_OFF_MANUAL_REQUEST);
END_REGION

REGION Network 25: SWITCH ON GENERAL CONDITION HELP
   RUNG wire#powerrail
      Contact( #SWITCH_ON_MANUAL_REQUEST )
      I_Contact( #SWITCH_ON_GENERAL_CONDITIONS )
      Coil( #SWITCH_ON_GENERAL_CONDITION_HELP )
   END_RUNG
   // the same network as SCL:
   #SWITCH_ON_GENERAL_CONDITION_HELP := #SWITCH_ON_MANUAL_REQUEST AND NOT #SWITCH_ON_GENERAL_CONDITIONS;
END_REGION

REGION Network 26: SWITCH ON INITIAL CONDITION HELP
   RUNG wire#powerrail
      Contact( #SWITCH_ON_MANUAL_REQUEST )
      Contact( #SWITCH_ON_GENERAL_CONDITIONS )
      I_Contact( #SWITCH_ON_INITIAL_CONDITIONS )
      Coil( #SWITCH_ON_INITIAL_CONDITION_HELP )
   END_RUNG
   // the same network as SCL:
   #SWITCH_ON_INITIAL_CONDITION_HELP := #SWITCH_ON_MANUAL_REQUEST AND #SWITCH_ON_GENERAL_CONDITIONS AND NOT #SWITCH_ON_INITIAL_CONDITIONS;
END_REGION

REGION Network 27: SWITCH OFF GENERAL CONDITION HELP
   RUNG wire#powerrail
      Contact( #SWITCH_OFF_MANUAL_REQUEST )
      I_Contact( #SWITCH_OFF_GENERAL_CONDITIONS )
      Coil( #SWITCH_OFF_GENERAL_CONDITION_HELP )
   END_RUNG
   // the same network as SCL:
   #SWITCH_OFF_GENERAL_CONDITION_HELP := #SWITCH_OFF_MANUAL_REQUEST AND NOT #SWITCH_OFF_GENERAL_CONDITIONS;
END_REGION

REGION Network 28: SWITCH OFF INITIAL CONDITION HELP
   RUNG wire#powerrail
      Contact( #SWITCH_OFF_MANUAL_REQUEST )
      Contact( #SWITCH_OFF_GENERAL_CONDITIONS )
      I_Contact( #SWITCH_OFF_INITIAL_CONDITIONS )
      Coil( #SWITCH_OFF_INITIAL_CONDITION_HELP )
   END_RUNG
   // the same network as SCL:
   #SWITCH_OFF_INITIAL_CONDITION_HELP := #SWITCH_OFF_MANUAL_REQUEST AND #SWITCH_OFF_GENERAL_CONDITIONS AND NOT #SWITCH_OFF_INITIAL_CONDITIONS;
END_REGION

REGION Network 29: HMI STATUS
   RUNG wire#powerrail
      Contact( "M_ONE" )
      wire#w1
      Contact( #OUT_OF_SERVICE )
      Coil( #HMI_POWER_UP_COND_OFF )
   END_RUNG
   RUNG wire#w1
      Contact( #IN_SERVICE )
      Coil( #HMI_POWER_UP_COND_ON )
   END_RUNG
   // the same network as SCL:
   #HMI_POWER_UP_COND_OFF := "M_ONE" AND #OUT_OF_SERVICE;
   #HMI_POWER_UP_COND_ON := "M_ONE" AND #IN_SERVICE;
END_REGION

REGION Network 30: HMI STATUS
   RUNG wire#powerrail
      Contact( "DB2001_MODES_GENERAL".GENERAL.MANUAL_SELECTED )
      wire#w1
      Contact( #SWITCH_OFF_GENERAL_CONDITIONS )
      Contact( #SWITCH_OFF_INITIAL_CONDITIONS )
      I_Contact( #OUT_OF_SERVICE )
      Coil( #HMI_POWER_UP_EXECU_LEFT )
   END_RUNG
   RUNG wire#w1
      Contact( #SWITCH_ON_GENERAL_CONDITIONS )
      Contact( #SWITCH_ON_INITIAL_CONDITIONS )
      I_Contact( #IN_SERVICE )
      Coil( #HMI_POWER_UP_EXECU_RIGHT )
   END_RUNG
   // the same network as SCL:
   #HMI_POWER_UP_EXECU_LEFT := "DB2001_MODES_GENERAL".GENERAL.MANUAL_SELECTED AND #SWITCH_OFF_GENERAL_CONDITIONS AND #SWITCH_OFF_INITIAL_CONDITIONS AND NOT #OUT_OF_SERVICE;
   #HMI_POWER_UP_EXECU_RIGHT := "DB2001_MODES_GENERAL".GENERAL.MANUAL_SELECTED AND #SWITCH_ON_GENERAL_CONDITIONS AND #SWITCH_ON_INITIAL_CONDITIONS AND NOT #IN_SERVICE;
END_REGION

REGION Network 31: MAIN VALVE OUTPUT
   RUNG wire#powerrail
      Contact( #SWITCH_ON )
      Coil( #MAIN_VALVE )
   END_RUNG
   // the same network as SCL:
   #MAIN_VALVE := #SWITCH_ON;
END_REGION
END_FUNCTION_BLOCK
